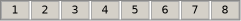
VISUALIZATION V_dwBitToggle  // 241x21
VAR_INPUT
  iNumOfCh : INT;
END_VAR
VAR_IN_OUT
	dwVar : DWORD;
END_VAR
    Rectangle (1,1 28x18), "1", colour toggle: dwVar.1, invisible if: iNumOfCh < 1
        toggle dwVar.1
    Rectangle (31,1 28x18), "2", colour toggle: dwVar.2, invisible if: iNumOfCh < 2
        toggle dwVar.2
    Rectangle (61,1 28x18), "3", colour toggle: dwVar.3, invisible if: iNumOfCh < 3
        toggle dwVar.3
    Rectangle (91,1 28x18), "4", colour toggle: dwVar.4, invisible if: iNumOfCh < 4
        toggle dwVar.4
    Rectangle (121,1 28x18), "5", colour toggle: dwVar.5, invisible if: iNumOfCh < 5
        toggle dwVar.5
    Rectangle (151,1 28x18), "6", colour toggle: dwVar.6, invisible if: iNumOfCh < 6
        toggle dwVar.6
    Rectangle (181,1 28x18), "7", colour toggle: dwVar.7, invisible if: iNumOfCh < 7
        toggle dwVar.7
    Rectangle (211,1 28x18), "8", colour toggle: dwVar.8, invisible if: iNumOfCh < 8
        toggle dwVar.8
END_VISUALIZATION

(* stored: Version 1.1.0.1, ProductVersion 3.1.4018.10
   Visu V_dwBitToggle: Id {5d46a79c-28a8-4ae9-ab64-1f3a7a18cdbe} *)
